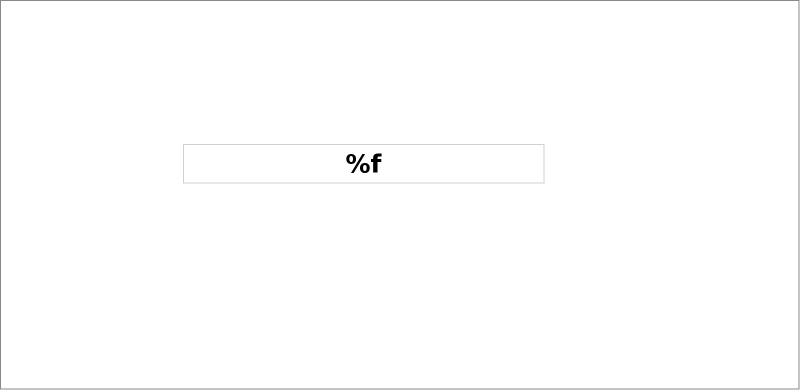
VISUALIZATION VisuEncoderInput  // 800x390
VAR_IN_OUT
	pDev : POINTER TO FB_EncoderBase;
END_VAR
    Textfield (183,144 361x39), "%f", text variable: pDev^.nOutPosition
END_VISUALIZATION

(* stored: Version 1.1.0.1, ProductVersion 3.1.4024.11
   Visu VisuEncoderInput: Id {bee66759-eebe-00ae-2627-bdba286735d8} *)
